{attribute addProperty BoxType "EK1100-0000-0018"}
{attribute addProperty Id "Beckhoff_EKxxxx_0080EK1122Beckhoff_EKxxxx_0080EK1122_49C116CC162A_0006_EK1122_0080_0019EK1122_179A0949162A_0005_EK1122_0080_0018EK1122_179A0949162A_0004_EK1122_0080_0017EK1122_179A0949162"}
{attribute addProperty CRC "4175618236"}
{attribute addProperty SizeInBites "64"}
{attribute addProperty SizeInBytes "8"}
TYPE Beckhoff_EKxxxx_0080_F8E2E0BC EXTENDS EK1100_179A0949 :
STRUCT
	{attribute addProperty Name "Beckhoff_EKxxxx_0080EK1122"}
	Beckhoff_EKxxxx_0080EK1122 : Beckhoff_EKxxxx_0080EK1122_49C116CC;
	{attribute addProperty Name "A_0006_EK1122_0080_0019"}
	A_0006_EK1122_0080_0019 : EK1122_179A0949;
	{attribute addProperty Name "A_0005_EK1122_0080_0018"}
	A_0005_EK1122_0080_0018 : EK1122_179A0949;
	{attribute addProperty Name "A_0004_EK1122_0080_0017"}
	A_0004_EK1122_0080_0017 : EK1122_179A0949;
END_STRUCT
END_TYPE

(* stored: Version 1.2.0.0, ProductVersion 3.1.4024.9
   DUT Beckhoff_EKxxxx_0080_F8E2E0BC: Id {d573e6d1-143b-4cdd-95c0-f36b52214186} *)
